Omron Sysmac Studio project Connect4Finishedbutcanbeautifymore (Sysmac Studio 1.56.0.64011, StandardProject)

# Controller new_Controller_0: NJ501-1500 version 1.64
Units and slaves: Power Supply : NJ-Px3001; CPU : NJ501-1500
Task PrimaryTask (priority 4, period or condition 1000): Program0

VAR_GLOBAL
    col : INT := 0;
    row : INT := 0;
    Board : ARRAY[1..7,1..6] OF INT;
    GameRunning : BOOL := True;
    ColumnSelected : INT := -1;
    CurrentPlayer : INT := 1;
    Winner : INT := 0;
    IsFull : BOOL := False;
    Index : INT := 0;
    Column : INT := 0;
    TempFull : BOOL := False;
    ColumnButton : ARRAY[0..7] of BOOL;
    RestartButton : BOOL := False;
    ValidMove : BOOL := False;
    DisplayText : STRING[255] := 'Welcome to Connect4';
END_VAR

PROGRAM Program0
VAR
    i : INT;
END_VAR
VAR_EXTERNAL
    col : INT;
    row : INT;
    Board : ARRAY[1..7,1..6] OF INT;
    GameRunning : BOOL;
    ColumnSelected : INT;
    CurrentPlayer : INT;
    Winner : INT;
    IsFull : BOOL;
    Index : INT;
    Column : INT;
    TempFull : BOOL;
    ColumnButton : ARRAY[0..7] of BOOL;
    RestartButton : BOOL;
    ValidMove : BOOL;
    DisplayText : STRING[255];
END_VAR

(* Section Section0: ladder, written here as Structured Text *)

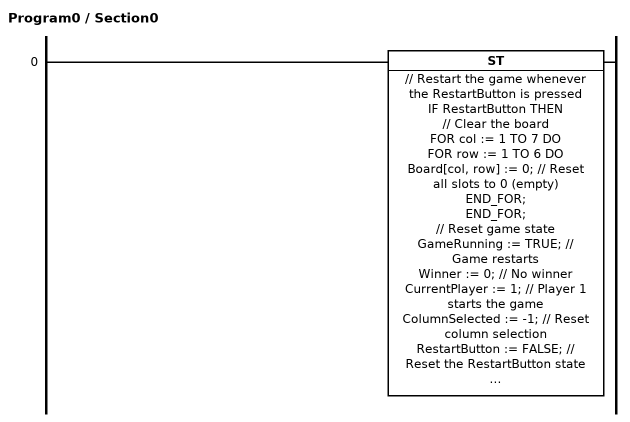
(* Rung 0 *)
// Restart the game whenever the RestartButton is pressed
IF RestartButton THEN
    // Clear the board
    FOR col := 1 TO 7 DO
        FOR row := 1 TO 6 DO
            Board[col, row] := 0; // Reset all slots to 0 (empty)
        END_FOR;
    END_FOR;

    // Reset game state
    GameRunning := TRUE; // Game restarts
    Winner := 0; // No winner
    CurrentPlayer := 1; // Player 1 starts the game
    ColumnSelected := -1; // Reset column selection
    RestartButton := FALSE; // Reset the RestartButton state
    ValidMove := FALSE; // Ensure no pending moves are tracked
	DisplayText := 'Welcome to Connect4';
	

    // Exit the game loop to immediately reset
    RETURN; // Ensures no further game logic executes after reset
END_IF;

// Main game loop
WHILE GameRunning DO

	// Restart the game whenever the RestartButton is pressed
IF RestartButton THEN
    // Clear the board
	
    FOR col := 1 TO 7 DO
        FOR row := 1 TO 6 DO
            Board[col, row] := 0; // Reset all slots to 0 (empty)
        END_FOR;
    END_FOR;

    // Reset game state
    GameRunning := TRUE; // Game restarts
    Winner := 0; // No winner
    CurrentPlayer := 1; // Player 1 starts the game
    ColumnSelected := -1; // Reset column selection
    RestartButton := FALSE; // Reset the RestartButton state
    ValidMove := FALSE; // Ensure no pending moves are tracked

    // Exit the game loop to immediately reset
    RETURN; // Ensures no further game logic executes after reset
END_IF;
	
    // Detect button press and set ColumnSelected
    FOR col := 1 TO 7 DO
        IF ColumnButton[col] THEN
            ColumnSelected := col; // Set selected column
            ColumnButton[col] := FALSE; // Reset button state
            EXIT; // Exit loop after detecting button press
        END_IF;
    END_FOR;

    // Drop the token into the lowest available slot in the selected column
    ValidMove := FALSE; // Variable to track if a valid move was made
    IF ColumnSelected >= 1 AND ColumnSelected <= 7 THEN
        FOR row := 6 TO 1 BY -1 DO // Start from the bottom row
            IF Board[ColumnSelected, row] = 0 THEN
                Board[ColumnSelected, row] := CurrentPlayer; // Place the token
                ValidMove := TRUE; // Mark the move as valid
                ColumnSelected := -1; // Reset column selection
                EXIT; // Stop after placing the token
            END_IF;
        END_FOR;
    END_IF;

    // Check for win condition
    FOR col := 1 TO 7 DO
        FOR row := 1 TO 6 DO
            // Check horizontal
            IF col <= 4 THEN
                IF Board[col, row] = CurrentPlayer AND
                   Board[col+1, row] = CurrentPlayer AND
                   Board[col+2, row] = CurrentPlayer AND
                   Board[col+3, row] = CurrentPlayer THEN
                    Winner := CurrentPlayer;
                    GameRunning := FALSE;
                END_IF;
            END_IF;

            // Check vertical
            IF row <= 3 THEN
                IF Board[col, row] = CurrentPlayer AND
                   Board[col, row+1] = CurrentPlayer AND
                   Board[col, row+2] = CurrentPlayer AND
                   Board[col, row+3] = CurrentPlayer THEN
                    Winner := CurrentPlayer;
                    GameRunning := FALSE;
                END_IF;
            END_IF;

            // Check diagonal (\ direction)
            IF col <= 4 AND row <= 3 THEN
                IF Board[col, row] = CurrentPlayer AND
                   Board[col+1, row+1] = CurrentPlayer AND
                   Board[col+2, row+2] = CurrentPlayer AND
                   Board[col+3, row+3] = CurrentPlayer THEN
                    Winner := CurrentPlayer;
                    GameRunning := FALSE;
                END_IF;
            END_IF;

            // Check diagonal (/ direction)
            IF col >= 4 AND row <= 3 THEN
                IF Board[col, row] = CurrentPlayer AND
                   Board[col-1, row+1] = CurrentPlayer AND
                   Board[col-2, row+2] = CurrentPlayer AND
                   Board[col-3, row+3] = CurrentPlayer THEN
                    Winner := CurrentPlayer;
                    GameRunning := FALSE;
                END_IF;
            END_IF;
        END_FOR;
    END_FOR;

    // Check for tie condition (board full)
    IsFull := TRUE;
    FOR col := 1 TO 7 DO
        IF Board[col, 1] = 0 THEN // Check the top row of each column
            IsFull := FALSE; // If there's an empty space, it's not a tie
            EXIT;
        END_IF;
    END_FOR;

    IF IsFull AND Winner = 0 THEN
        GameRunning := FALSE; // End the game as a tie
    END_IF;

    // Switch players only if a valid move was made
    IF Winner = 0 AND ValidMove THEN
        IF CurrentPlayer = 1 THEN
            CurrentPlayer := 2; // Switch to Player 2
        ELSE
            CurrentPlayer := 1; // Switch to Player 1
        END_IF;
    END_IF;
	
	    IF (Winner <> 0) THEN
        IF Winner = 1 THEN
            DisplayText := 'Player 1 Wins!';
        ELSIF Winner = 2 THEN
            DisplayText := 'Player 2 Wins!';
        END_IF;
    ELSIF (IsFull = TRUE) THEN
        // We found a draw condition
        DisplayText := 'It is a Draw!';
    END_IF;

END_WHILE;
END_PROGRAM

# Device HMI_NA5_0 (NA): not converted